// TIA Portal V19 export
FUNCTION "MeasWheelCheckRotation_TypeEnc2" : Int   // FC50, LAD
TITLE = Check velocity of the measuring wheel compared with axis (motor) command
// Da usare con encoder rotella di misura su secondo encoder dell'asse di posizionamento e velocità di confronto che è esterna (esempio la raddrizzatrice spinge il  materiale dentro all'alimentatore a rulli che è aperto e quindi non muove lui stesso la lamiera) oppure è la velocità dell'asse in anello aperto (ad esempio l'alimentatore a rulli chiuso che muove la lamiera).
// stored: Access Published, SetENOAutomatically false
   VAR_INPUT
      TO_Ax : TO_PositioningAxis;
      VelMaterialMover : LReal;   // "#TO_Ax.Velocity" of extrenal material mover that move the Meas Wheel
      VelMin : LReal;   // Min velocity for execute check
      ErrPercentageMax : LReal;   // Max error % beetween velocity
   END_VAR
   VAR_OUTPUT
      Err : LReal;   // Show % actual error percentage
   END_VAR
   VAR_TEMP
      MeasWheelIsActive : Bool;
      MotorVelocity : LReal;
      MotorVelocityABS : LReal;
      ErrorPercentage : LReal;
      Check : Bool;
   END_VAR
   VAR CONSTANT
      RET_NULL : Int := 0;
      RET_VEL_OK : Int := 1;
      RET_VEL_BELOW_MIN : Int := 10;
      RET_ERR_ENC_NOT_VALID : Int := 101;
      RET_VEL_DELTA_EXCEED : Int := 103;
   END_VAR
   VAR_TEMP   // added for the SCL form of the ladder/FBD networks
      _w1 : Bool;
   END_VAR
BEGIN

REGION Network 1: Out error percentage
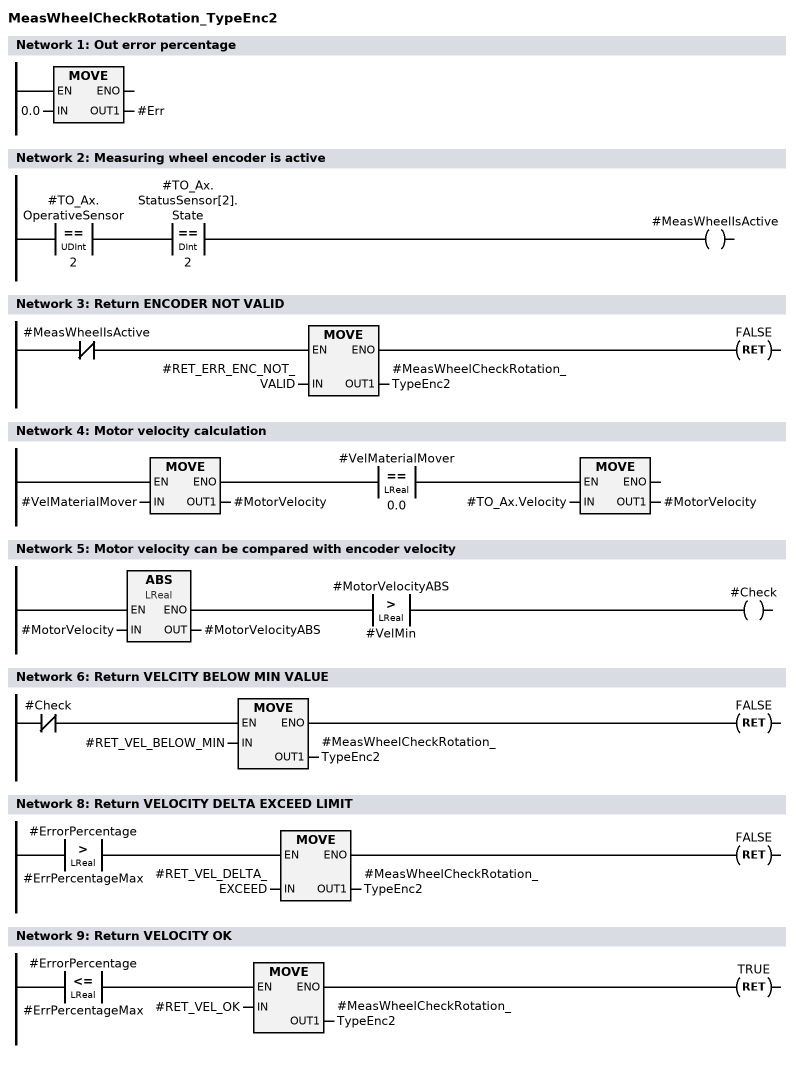
   RUNG wire#powerrail
      { S7_GenerateENO := "TRUE" } Move(in := 0.0, out1 => #Err)
   END_RUNG
   // the same network as SCL:
   #Err := 0.0;
END_REGION

REGION Network 2: Measuring wheel encoder is active
   RUNG wire#powerrail
      { S7_Templates := "SrcType := UDInt" } EQ_Contact(in1 := #TO_Ax.OperativeSensor, in2 := 2)
      { S7_Templates := "SrcType := DInt" } EQ_Contact(in1 := #TO_Ax.StatusSensor[2].State, in2 := 2)
      Coil( #MeasWheelIsActive )
   END_RUNG
   // the same network as SCL:
   #MeasWheelIsActive := (#TO_Ax.OperativeSensor = 2) AND (#TO_Ax.StatusSensor[2].State = 2);
END_REGION

REGION Network 3: Return ENCODER NOT VALID
   RUNG wire#powerrail
      I_Contact( #MeasWheelIsActive )
      { S7_GenerateENO := "TRUE" } Move(in := #RET_ERR_ENC_NOT_VALID, out1 => #MeasWheelCheckRotation_TypeEnc2)
      ReturnCoil( FALSE )
   END_RUNG
   // the same network as SCL:
   // ENO of a box is taken as its EN; it also drops when the box reports an error
   IF NOT #MeasWheelIsActive THEN
       #MeasWheelCheckRotation_TypeEnc2 := #RET_ERR_ENC_NOT_VALID;
       ENO := FALSE;
       RETURN;
   END_IF;
END_REGION

REGION Network 4: Motor velocity calculation
   RUNG wire#powerrail
      { S7_GenerateENO := "TRUE" } Move(in := #VelMaterialMover, out1 => #MotorVelocity)
      { S7_Templates := "SrcType := LReal" } EQ_Contact(in1 := #VelMaterialMover, in2 := 0.0)
      { S7_GenerateENO := "TRUE" } Move(in := #TO_Ax.Velocity, out1 => #MotorVelocity)
   END_RUNG
   // the same network as SCL:
   // ENO of a box is taken as its EN; it also drops when the box reports an error
   #MotorVelocity := #VelMaterialMover;
   IF #VelMaterialMover = 0.0 THEN #MotorVelocity := #TO_Ax.Velocity; END_IF;
END_REGION

REGION Network 5: Motor velocity can be compared with encoder velocity
   RUNG wire#powerrail
      { S7_Templates := "SrcType := LReal"; S7_GenerateENO := "TRUE" } Abs(in := #MotorVelocity, out => #MotorVelocityABS)
      { S7_Templates := "SrcType := LReal" } GT_Contact(in1 := #MotorVelocityABS, in2 := #VelMin)
      Coil( #Check )
   END_RUNG
   // the same network as SCL:
   // ENO of a box is taken as its EN; it also drops when the box reports an error
   #MotorVelocityABS := ABS(#MotorVelocity);
   #Check := #MotorVelocityABS > #VelMin;
END_REGION

REGION Network 6: Return VELCITY BELOW MIN VALUE
   RUNG wire#powerrail
      I_Contact( #Check )
      { S7_GenerateENO := "TRUE" } Move(in := #RET_VEL_BELOW_MIN, out1 => #MeasWheelCheckRotation_TypeEnc2)
      ReturnCoil( FALSE )
   END_RUNG
   // the same network as SCL:
   // ENO of a box is taken as its EN; it also drops when the box reports an error
   IF NOT #Check THEN
       #MeasWheelCheckRotation_TypeEnc2 := #RET_VEL_BELOW_MIN;
       ENO := FALSE;
       RETURN;
   END_IF;
END_REGION

REGION Network 7 (SCL): Error percentale between motor and encoder

   #ErrorPercentage := ABS(100.0 * (#TO_Ax.StatusExtrapolation.ExtrapolatedVelocity - #MotorVelocity) / #MotorVelocity);

   #Err := #ErrorPercentage;
END_REGION

REGION Network 8: Return VELOCITY DELTA EXCEED LIMIT
   RUNG wire#powerrail
      { S7_Templates := "SrcType := LReal" } GT_Contact(in1 := #ErrorPercentage, in2 := #ErrPercentageMax)
      { S7_GenerateENO := "TRUE" } Move(in := #RET_VEL_DELTA_EXCEED, out1 => #MeasWheelCheckRotation_TypeEnc2)
      ReturnCoil( FALSE )
   END_RUNG
   // the same network as SCL:
   // ENO of a box is taken as its EN; it also drops when the box reports an error
   #_w1 := #ErrorPercentage > #ErrPercentageMax;
   IF #_w1 THEN
       #MeasWheelCheckRotation_TypeEnc2 := #RET_VEL_DELTA_EXCEED;
       ENO := FALSE;
       RETURN;
   END_IF;
END_REGION

REGION Network 9: Return VELOCITY OK
   RUNG wire#powerrail
      { S7_Templates := "SrcType := LReal" } LE_Contact(in1 := #ErrorPercentage, in2 := #ErrPercentageMax)
      { S7_GenerateENO := "TRUE" } Move(in := #RET_VEL_OK, out1 => #MeasWheelCheckRotation_TypeEnc2)
      ReturnCoil( TRUE )
   END_RUNG
   // the same network as SCL:
   // ENO of a box is taken as its EN; it also drops when the box reports an error
   #_w1 := #ErrorPercentage <= #ErrPercentageMax;
   IF #_w1 THEN
       #MeasWheelCheckRotation_TypeEnc2 := #RET_VEL_OK;
       ENO := TRUE;
       RETURN;
   END_IF;
END_REGION
END_FUNCTION
